FUNCTION_BLOCK Axis_Base IMPLEMENTS I_AxisBase, I_Axis, I_Position, I_Status, I_Velocity, I_Jog, I_Object, I_Cyclic, I_Resettable
VAR
	_axis : REFERENCE TO Tc2_MC2.AXIS_REF;
	EnableBehaviour : EnableDisableTask;
	DefaultResetBehaviour : CoEResetTask;
	DefaultMoveBehaviour : MoveAbsTask;
	DefaultRelBehaviour : MoveRelTask;
	DefaultModBehaviour : MoveModTask;
	DefaultVeloBehaviour : MoveVeloTask;
	DefaultJogBehaviour : JogTask;
	HaltBehaviour	: HaltTask;
	TaskCollection : ObjectRunner<99>;
	axesReadError : Tc2_MC2.MC_ReadAxisError;
	_ErrorId: DWORD;
	DemandVelo : LREAL;
END_VAR

{analysis -2}

PROPERTY PUBLIC Acceleration : mc_lreal
GET
Acceleration := DefaultMoveBehaviour.Acceleration;
END_GET
SET
DefaultMoveBehaviour.Acceleration := Acceleration;
END_SET
END_PROPERTY

PROPERTY AxisRef : reference to Axis_Ref
GET
AxisRef REF= _axis;
END_GET
END_PROPERTY

PROPERTY BufferMode : MC_BufferMode
GET
BufferMode := DefaultMoveBehaviour.BufferMode;
END_GET
SET
DefaultMoveBehaviour.BufferMode:= BufferMode;
DefaultRelBehaviour.BufferMode := BufferMode;
DefaultModBehaviour.BufferMode := BufferMode;
END_SET
END_PROPERTY

PROPERTY CurrentPosition : LREAL
GET
CurrentPosition := _axis.NcToPlc.ActPos;
END_GET
END_PROPERTY

PROPERTY CurrentVelocity : LREAL
GET
CurrentVelocity := _axis.NcToPlc.ActVelo;
END_GET
END_PROPERTY

METHOD Cycle : HRESULT
VAR_INPUT
END_VAR
_axis.ReadStatus();
axesReadError(Axis := _axis, Enable := TRUE, AxisErrorID => _ErrorId);
TaskCollection.Cycle();
END_METHOD

PROPERTY PUBLIC Deceleration : mc_lreal
GET
Deceleration := DefaultMoveBehaviour.Deceleration;
END_GET
SET
DefaultMoveBehaviour.Deceleration := Deceleration;
HaltBehaviour.Deceleration := Deceleration;
END_SET
END_PROPERTY

METHOD PUBLIC DisableAxis : HRESULT
VAR_INPUT
END_VAR
DisableAxis := EnableBehaviour.Disable();
END_METHOD

METHOD PUBLIC EnableAxis : HRESULT
VAR_INPUT
	InhibitPositive : BOOL;
	InhibitNegative : BOOL;
END_VAR
EnableBehaviour.InhibitNegative := InhibitNegative;
EnableBehaviour.InhibitPositive := InhibitPositive;
EnableAxis := EnableBehaviour.Enable();
END_METHOD

PROPERTY ErrorID : DWORD
GET
ErrorId := _ErrorId;
END_GET
END_PROPERTY

//FB_Init is always available implicitly and it is used primarily for initialization.
//The return value is not evaluated. For a specific influence, you can also declare the
//methods explicitly and provide additional code there with the standard initialization
//code. You can evaluate the return value.
METHOD FB_Init: BOOL
VAR_INPUT
    bInitRetains: BOOL; // TRUE: the retain variables are initialized (reset warm / reset cold)
    bInCopyCode: BOOL;  // TRUE: the instance will be copied to the copy code afterward (online change) 
	Axis : Reference TO AXIS_REF;  
END_VAR
EnableBehaviour.AxisRef REF= axis;
DefaultResetBehaviour.AxisRef REF= axis;
DefaultMoveBehaviour.AxisRef REF= axis;
DefaultVeloBehaviour.AxisRef REF= axis;
DefaultJogBehaviour.AxisRef REF= axis;
DefaultRelBehaviour.AxisRef REF= axis;
DefaultModBehaviour.AxisRef REF= axis;
HaltBehaviour.AxisRef REF= axis;
_axis REF= Axis;

DefaultJogBehaviour.RegisterWithParent(Parent := TaskCollection);
DefaultModBehaviour.RegisterWithParent(Parent := TaskCollection);
DefaultMoveBehaviour.RegisterWithParent(Parent := TaskCollection);
DefaultRelBehaviour.RegisterWithParent(Parent := TaskCollection);
DefaultJogBehaviour.RegisterWithParent(Parent := TaskCollection);
DefaultVeloBehaviour.RegisterWithParent(Parent := TaskCollection);
HaltBehaviour.RegisterWithParent(Parent := TaskCollection);
DefaultResetBehaviour.RegisterWithParent(Parent := TaskCollection);
EnableBehaviour.RegisterWithParent(Parent := TaskCollection);
END_METHOD

METHOD PUBLIC HaltAxis : HRESULT
VAR
END_VAR
IF NOT HaltBehaviour.Busy THEN
	HaltAxis := HaltBehaviour.Execute();
	DefaultMoveBehaviour.Abort();
	DefaultVeloBehaviour.Abort();
ELSE 
	HaltAxis := -1;
END_IF
END_METHOD

PROPERTY HasError : BOOL
GET
HasError := _axis.Status.Error;
END_GET
END_PROPERTY

METHOD Inch : HRESULT
VAR_INPUT
	Distance : MC_LREAL;
	Direction : BOOL;
END_VAR
IF FAILED( DefaultJogBehaviour.Inch(Distance, Direction)) THEN
	Inch := -1;
END_IF
END_METHOD

PROPERTY InTargetPosition : BOOL
GET
InTargetPosition := _axis.Status.InTargetPosition;
END_GET
END_PROPERTY

PROPERTY InVelocity : BOOL
GET
InVelocity := ABS(_axis.NcToPlc.ActVelo) < DemandVelo + (DemandVelo * 0.02) AND 
				ABS(_axis.NcToPlc.ActVelo) > DemandVelo - (DemandVelo * 0.02);
END_GET
END_PROPERTY

PROPERTY IsCoupled : bool
GET
isCoupled := _axis.Status.Coupled;
END_GET
END_PROPERTY

PROPERTY IsEnabled : bool
GET
isEnabled := not _axis.Status.Disabled;
END_GET
END_PROPERTY

PROPERTY IsStationary : bool
GET
isStationary := _axis.NcToPlc.SetVelo = 0;
END_GET
END_PROPERTY

PROPERTY PUBLIC Jerk : mc_lreal
GET
Jerk := DefaultMoveBehaviour.Jerk;
END_GET
SET
DefaultMoveBehaviour.Jerk := Jerk;
HaltBehaviour.Jerk := Jerk;
END_SET
END_PROPERTY

METHOD JogFast : HRESULT
VAR_INPUT
	Direction : BOOL;
END_VAR
IF FAILED(DefaultJogBehaviour.JogFast(Direction)) THEN
	JogFast := -1;
END_IF
END_METHOD

METHOD JogSlow : HRESULT
VAR_INPUT
	Direction : BOOL;
END_VAR
IF FAILED(DefaultJogBehaviour.JogSlow(Direction)) THEN
	JogSlow := -1;
END_IF
END_METHOD

METHOD MoveAtVelocity : HRESULT
VAR_INPUT
	Direction : MC_Direction;
	Velocity : MC_LREAL;
END_VAR
IF Velocity = 0 THEN 
	MoveAtVelocity := -1;
	RETURN;
END_IF

IF SUCCEEDED(DefaultVeloBehaviour.MoveAtVelocity(Direction, Velocity)) THEN
	DemandVelo := Velocity;
ELSE
	MoveAtVelocity := -1;
END_IF
END_METHOD

METHOD MoveByDistance : HRESULT
VAR_INPUT
	Distance : MC_LREAL;
	Velocity : MC_LREAL;
END_VAR
IF ABS(Distance) = 0 THEN
	MoveByDistance := -1;
	RETURN;
END_IF
IF _axis.Status.Disabled THEN
	MoveByDistance := -2;
	RETURN;
END_IF

IF _axis.Status.Error THEN
	MoveByDistance := -3;
	RETURN;
END_IF

DefaultRelBehaviour.MoveBy(Distance,Velocity);
END_METHOD

METHOD MoveToModuloPosition : HRESULT
VAR_INPUT
	Position : MC_LREAL;
	Velocity : MC_LREAL;
END_VAR
IF Velocity = 0 THEN
	MoveToModuloPosition := -1;
	RETURN;
END_IF

IF _axis.Status.Disabled THEN
	MoveToModuloPosition := -2;
	RETURN;
END_IF

IF _axis.Status.Error THEN
	MoveToModuloPosition := -3;
	RETURN;
END_IF

DefaultModBehaviour.MoveTo(Position,Velocity);
END_METHOD

METHOD PUBLIC MoveToPosition : HRESULT
VAR_INPUT
	Position : MC_LREAL;
	Velocity : MC_LREAL;
END_VAR
IF Velocity = 0 THEN
	MoveToPosition := -1;
	RETURN;
END_IF

IF _axis.Status.Disabled THEN
	MoveToPosition := -2;
	RETURN;
END_IF

IF _axis.Status.Error THEN
	MoveToPosition := -3;
	RETURN;
END_IF

DefaultMoveBehaviour.MoveTo(Position,Velocity);
END_METHOD

METHOD RegisterWithParent
VAR_INPUT
	Parent	: Base_Library.I_HostObjects;
END_VAR
Parent.RegisterCyclic(THIS^);
Parent.RegisterResettable(THIS^);
END_METHOD

METHOD PUBLIC Reset : HRESULT
VAR
	ResetResult : HRESULT;
	MoveAbortResult : BOOL;
	HaltAbortResult : BOOL;
END_VAR
TaskCollection.Reset();
//TaskCollection.Abort();
END_METHOD

END_FUNCTION_BLOCK

(* stored: Version 1.1.0.1
   POU Axis_Base: Id {6091fbf5-8563-4c3d-a46f-a871d52562e9}, SpecialFunc None
   Folder Base: Id {bc93d43c-3186-404b-ac84-315fffe3aac4}
   Folder Dynamics: Id {cb4086e9-6981-4aa8-9a87-7a24dd3c8528}
   Folder Manual: Id {9d120552-2d62-4889-ac32-0f0c4ddbbd86}
   Folder Position: Id {b9c6e694-8906-4efb-bd9d-8fd3dc8e33ad}
   Folder Status: Id {91eb89a1-3e50-4f9b-a3c9-6207bfd52c53}
   Folder Velocity: Id {d6f72365-77a8-427b-9fe5-df2e73a6c92a}
   Property Acceleration: Id {6323273a-3225-4f5a-9181-064e3eedda66}
   Get Get: Id {34764180-07ec-4ccd-a6b8-92e00db717a8}
   Set Set: Id {b780dd24-dc2c-4df0-8817-84480edf7b7e}
   Property AxisRef: Id {aaea047b-5e2b-4dbe-9bce-7ee41542008d}
   Get Get: Id {824cd367-141c-47b9-8e15-5709b4963377}
   Property BufferMode: Id {d08e2361-5203-4398-8c61-726e8a84e0a3}
   Get Get: Id {9e81ee1e-088d-4c14-a24d-933fb207a31e}
   Set Set: Id {520c3d3e-0864-445a-a57c-42fec43ce8ec}
   Property CurrentPosition: Id {f81022c8-aabe-4350-937c-d5e331c84e53}
   Get Get: Id {31d53272-f477-419f-9f8f-b2455c97ac7a}
   Property CurrentVelocity: Id {c88251f7-bef5-418d-9bae-83d23009f166}
   Get Get: Id {bc628771-a224-458b-b10f-81135cefb406}
   Method Cycle: Id {6e2b69ab-f1bf-4962-bdbb-f480f753daf6}
   Property Deceleration: Id {bb54abe4-e56a-4330-9f3c-f7af329a7f17}
   Get Get: Id {433beca3-2b49-4ba6-9d63-f01118a89332}
   Set Set: Id {28be4d06-067d-435d-89a3-c0ee8fd02e9d}
   Method DisableAxis: Id {4ca2c35a-d664-47dd-b699-e212d5be22eb}
   Method EnableAxis: Id {a835c18f-6175-4614-a6ac-65491f5fc70d}
   Property ErrorID: Id {23aaf61d-867b-4a0d-829f-c516b080f5fb}
   Get Get: Id {1db8f21e-3bb5-4924-ba79-9b04f8a9157c}
   Method FB_Init: Id {b79a0e62-0ee6-47b6-874a-a1e2579a6c1b}
   Method HaltAxis: Id {b5b4d676-a559-4d25-8571-0c2ec9c3c015}
   Property HasError: Id {a508d66e-2c23-49e5-bf01-8d54382ab174}
   Get Get: Id {26e58127-3309-47b3-91dd-05ea60bb0e3f}
   Method Inch: Id {a8ecae9a-5934-4e49-93bc-ed8a7c89528c}
   Property InTargetPosition: Id {9abca603-e884-4f4f-bccc-fc41fc8ff5ee}
   Get Get: Id {25924b82-ccca-4ae9-aec4-bfae0b30c843}
   Property InVelocity: Id {58797bbc-1847-4345-b88d-e9a061a816ed}
   Get Get: Id {2d341fd7-f727-4430-a670-3040afdfb9d4}
   Property IsCoupled: Id {6b5c09b2-f69c-4bfa-8f55-e28d0dee4f96}
   Get Get: Id {5710167e-5ed2-4c8f-a7c3-1f2e8d1de119}
   Property IsEnabled: Id {61d475f5-477d-4a41-ac2b-c5e94d4efd87}
   Get Get: Id {c410a671-3e66-4117-ad8d-e6127a67edec}
   Property IsStationary: Id {c81c5586-ca5c-467c-9e94-5811eaa88ec6}
   Get Get: Id {ee3f5e21-c9c4-44e4-88f0-3b457286107f}
   Property Jerk: Id {79ff8a18-6bf8-46ba-a24c-7f84c4790e08}
   Get Get: Id {66a6c61c-9532-41a0-a772-02a7efa824e1}
   Set Set: Id {fce2a919-a42f-43d2-85c4-9447d205ce29}
   Method JogFast: Id {95cc0a16-a1bd-4e7f-963c-68820a459e0a}
   Method JogSlow: Id {6f896ef2-e375-4b54-96df-82c467e4828a}
   Method MoveAtVelocity: Id {6d3a50a7-ce83-4f3f-b972-fcb26bf76028}
   Method MoveByDistance: Id {957d5870-8bcd-44f2-a483-ac5c3f32f182}
   Method MoveToModuloPosition: Id {470f0d21-ab3e-4d10-948f-9938775e223b}
   Method MoveToPosition: Id {bca42834-4b90-4808-be50-ee67839e4111}
   Method RegisterWithParent: Id {381741fc-fc26-4603-bb08-86e14ada8bdb}
   Method Reset: Id {bd5b60f2-6a45-4850-931f-c2efbdee4a44} *)
